// TIA Portal V17 export
// export: Created 2024-08-07T21:44:15.5502355Z, ExportSetting WithDefaults, DisplayName Totally Integrated Automation Portal, DisplayVersion V17 Update 7, DisplayName TIA Portal Openness, DisplayVersion V17 Update 7, DisplayName TIA Portal Version Control Interface, DisplayVersion V17, DisplayName SINAMICS Startdrive Advanced, DisplayVersion V17 SP2, DisplayName SINAMICS Startdrive G110M, G120, G120C, G120D, G120P, G115D, DisplayVersion V17 SP2, DisplayName SINAMICS Startdrive G130, G150, S120, S150, SINAMICS MV, S210, DisplayVersion V17 SP2, DisplayName STEP 7 Professional, DisplayVersion V17 Update 7, DisplayName STEP 7 Safety, DisplayVersion V17 Update 6, DisplayName WinCC Advanced / Unified PC, DisplayVersion V17 Update 7
TYPE "UDT_FittingParameters"
// stored: IsFailsafeCompliant false
   STRUCT
      DigiforceProgram : Int;
      FinalSpeed : Real;
      ApproachSpeed : Real;
      FinalForce : Real;
      ApproachForce : Real;
      EndWayImmediate : Real;   // relative position from digiforce
      EndWayWithTimeout : Real;   // relative position from digiforce
      SwitchingWay : Real;   // absolute cylinder position
      EndWayTimeout : Time;
   END_STRUCT;
END_TYPE
